# EPICS substitutions: ek9000App/Db/EL4004.substitutions
file EL4004.template
{       pattern
        {
                TERMINAL,

        }
        {
        }
}
